TYPE ST_TestStruct2 :
STRUCT
	nested_variable : TIME;
END_STRUCT
END_TYPE

(* stored: Version 1.1.0.1, ProductVersion 3.1.4024.11
   DUT ST_TestStruct2: Id {d66b4b2e-12c5-4512-8608-a2d437a2e762} *)
